// Specify a 1D mouvement, the position only represents a point in the 1D space
TYPE MoveProfile1D_t EXTENDS MoveProfile_t:
STRUCT
    lrPosition  : LREAL;         // Position to go
END_STRUCT
END_TYPE

(* stored: Version 1.1.0.1, ProductVersion 3.1.4024.6
   DUT MoveProfile1D_t: Id {a927e1fc-73c5-41fa-ae1e-b1b2d2fe83ad} *)
